FUNCTION_BLOCK INTERNAL FB_LightTowerComponent IMPLEMENTS I_LightTowerComponent
VAR
	_state	: BOOL;
END_VAR

METHOD Activate
_state := TRUE;
END_METHOD

METHOD Deactivate
_state := FALSE;
END_METHOD

PROPERTY State : BOOL
GET
State := _state;
END_GET
END_PROPERTY

END_FUNCTION_BLOCK

(* stored: Version 1.1.0.1, ProductVersion 3.1.4024.13
   POU FB_LightTowerComponent: Id {41abef2b-3003-0d85-20a0-65e892e3520f}, SpecialFunc None
   Method Activate: Id {deeea55e-7220-0b94-367f-ca32b7d51667}
   Method Deactivate: Id {d9a89d88-6178-0842-21bd-0933fa4f573f}
   Property State: Id {e1dce7d0-4136-0860-28f7-95520acfe064}
   Get Get: Id {8cac2eda-eb36-0516-3277-a66b42136080} *)
